	FUNCTION_BLOCK FB 357
	TITLE =G257M COOLING / HEATING GERM 8
	//COPYRIGHT:    (C) 2009  BUHLER AG, CH-9240 UZWIL, SWITZERLAND
	//
	//PRODUCT:      WinCoS_BIW01_09
	//
	//TITLE:        COOLING / HEATING GERM 8
	//                Machine group control
	//                Maschinengruppensteuerung
	//
	//--------------------------------------------------------------------------------
	//
	//IDENT:        AUTHOR:             DEPT:                              DATE:
	//
	//P01_FB357.1.0 K.Renz              CSB41                              13.Jan.2010
	//             1st Release
	//
	//--------------------------------------------------------------------------------
	//
	//PURPOSE:
	//
	//MANUAL :
	//
	//RESTRICTIONS:
	//
	//--------------------------------------------------------------------------------
	AUTHOR  : KR
	FAMILY  : USW
	VERSION : 9.9


	VAR
	  Gr       : FB10;	//Standard interface to group
	  InOutValue1    : DINT; //Data for user
	  InOutValue2    : DINT; //Data for user
	  OutWayConflict : BOOL;	//Data for user
	  OutSelectionOk : BOOL;	//Data for user
	  CmdNewValue : BOOL;	//Data for user
	  CmdNewJob   : BOOL;	//Data for user
	  OutCodeOK   : BOOL;	//Data for user
	  InEndOfJob  : BOOL ;	//Data for user
	  staWayOk      : BOOL ;	//Data for user
	  EdgeStartRelease : BOOL ;	//Data for user
	  USW8  : BOOL;	//Data for user
	  USW9 : BOOL;	//Data for user
	  USW10: BOOL;	//Data for user
	  USW11: BOOL;	//Data for user
	  USW12: BOOL;	//Data for user
	  USW13: BOOL;	//Data for user
	  USW14: BOOL;	//Data for user
	  USW15: BOOL;	//Data for user
	     #A_2845_QXV21 : FB12;   // Motor
	     #A_2845_QXV21AI : FB19;   // AnaInp
	     #A_2845_QXV21AO : FB17;   // AnaOutp
	     #A_2845_QXV21I1 : FB14;   // DigInpCont
	     #A_2845_QXV21I2 : FB14;   // DigInpCont
	     #A_2845_QXV31 : FB12;   // Motor
	     #A_2845_QXV31AI : FB19;   // AnaInp
	     #A_2845_QXV31AO : FB17;   // AnaOutp
	     #A_2845_QXV31I1 : FB14;   // DigInpCont
	     #A_2845_QXV31I2 : FB14;   // DigInpCont
	     #A_2854_MXZ01 : FB12;   // Motor
	     #A_2855_MXZ01 : FB12;   // Motor
	END_VAR
	VAR_TEMP
	   tmpEnable		: BOOL;
	   tmpFlag  		: BOOL;
	   tmpCmdNext		: BOOL;
	   tmpLocal  		: BOOL;
	   tmpAspOk  		: BOOL;
	   tmpHWStop 		: BOOL;
	   tmpInstanzDBNo       : INT ;
	END_VAR
	BEGIN
	NETWORK
	TITLE =
	NETWORK
	TITLE =Read command from group control
	//Parameter
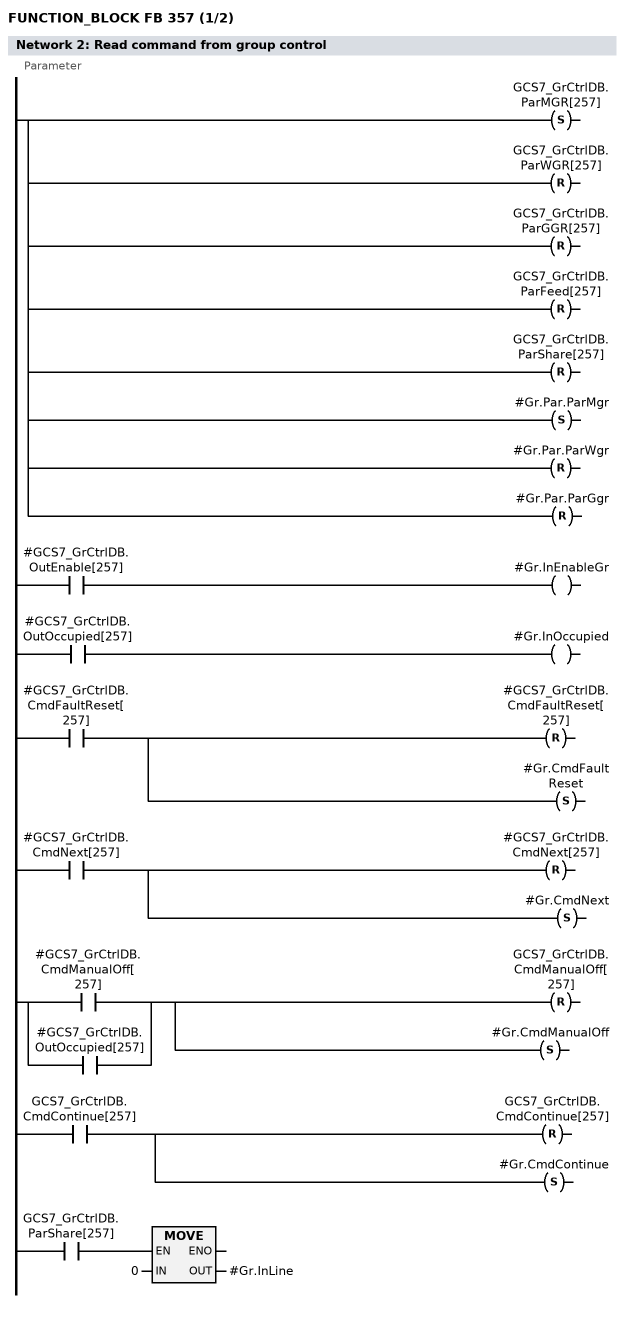
	      SET;
	      S   GCS7_GrCtrlDB.ParMGR[257];
	      R   GCS7_GrCtrlDB.ParWGR[257];
	      R   GCS7_GrCtrlDB.ParGGR[257];
	      R   GCS7_GrCtrlDB.ParFeed[257];
	      R   GCS7_GrCtrlDB.ParShare[257];
	      S   #Gr.Par.ParMgr;
	      R   #Gr.Par.ParWgr;
	      R   #Gr.Par.ParGgr;
	//Command
	      U   #GCS7_GrCtrlDB.OutEnable[257];
	      =   #Gr.InEnableGr;
	      U   #GCS7_GrCtrlDB.OutOccupied[257];
	      =   #Gr.InOccupied;
	      U   #GCS7_GrCtrlDB.CmdFaultReset[257];
	      R   #GCS7_GrCtrlDB.CmdFaultReset[257];
	      S   #Gr.CmdFaultReset;
	      U  #GCS7_GrCtrlDB.CmdNext[257];
	      R   #GCS7_GrCtrlDB.CmdNext[257];
	      S   #Gr.CmdNext;
	      U   #GCS7_GrCtrlDB.CmdManualOff[257];
	      O   #GCS7_GrCtrlDB.OutOccupied[257];
	      R   GCS7_GrCtrlDB.CmdManualOff[257];
	      S   #Gr.CmdManualOff;
	      U  GCS7_GrCtrlDB.CmdContinue[257];
	      R   GCS7_GrCtrlDB.CmdContinue[257];
	      S   #Gr.CmdContinue;
	//Init Line Number
	      U   GCS7_GrCtrlDB.ParShare[257];
	      SPBN WE00;
	      L     0;
	      T     #Gr.InLine;
	WE00: NOP   0;
	NETWORK
	TITLE =Call Methode Control
	// 1. Handle Interface PCControl
	// 2. Prepare mode --> ModePassive,ModeActive,ModeIdling
	// 3. Reset global flags of the group
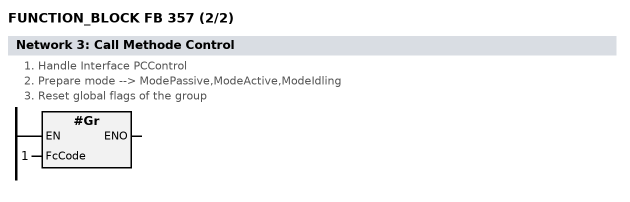
	      CALL #Gr (
	           FcCode                   := 1);
	NETWORK
	TITLE =Restart Idling Time
		L  #Gr.Par.ParIdling;
		L  2;
		>=I;
		SPB IdTm;
		T  #Gr.Par.ParIdling;
	IdTm:   NOP 0;
	      CLR;
	      S    #Gr.CmdRestartIdling;
	NETWORK
	TITLE =Prepare global flags
	NETWORK
	TITLE =Set Pattern (Target position)
	NETWORK
	TITLE =Interlocking WayOk
	//
	NETWORK
	TITLE =Interlocking Autostart
		CLR;
		R   #Gr.OutAutostart;
	NETWORK
	TITLE =Interlocking Enable
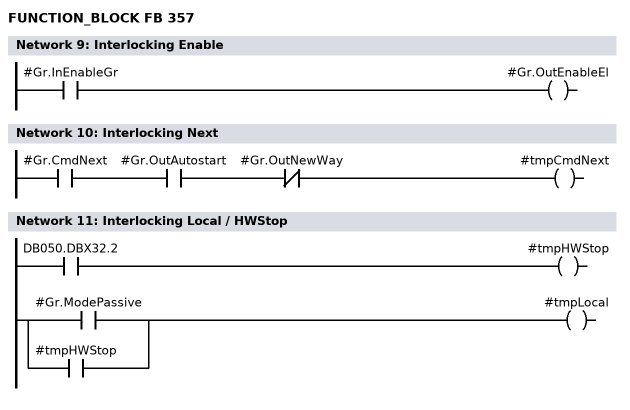
	      U     #Gr.InEnableGr;
	      =     #Gr.OutEnableEl;

	NETWORK
	TITLE =Interlocking Next
	      U     #Gr.CmdNext;
	      U     #Gr.OutAutostart;
	      UN    #Gr.OutNewWay;
	      =    #tmpCmdNext;

	NETWORK
	TITLE =Interlocking Local / HWStop
	      U    DB050.DBX32.2;
	      =    #tmpHWStop;

	      U    #Gr.ModePassive;
	      O    #tmpHWStop;
	      =    #tmpLocal;

	NETWORK
	TITLE =Interlocking Start Warning
	      NOP 0;
	//- Restart after fault --
	      U     #Gr.CmdFaultReset;
	      U     #Gr.VarFault;
	      S       "SYS_StartWarningDB".Area[9].CmdResetStartWarning;
	//- Run Timer --
	      AUF "G257M";
	      CALL  FB100 , DB100(
	       InModeHigher :=FALSE,
	       InArea     :=9,
	       InEnable   :=#Gr.OutEnableEl,
	       InLocal    :=#tmpLocal,
	       InStarted  :=#Gr.VarStarted,
	       InCmdNext  :=#tmpCmdNext,
	       OutCmdNext :=#tmpCmdNext,
	       OutStartwarning:=#Gr.VarStartWarning);
	//- Store Startwarning done  --
	//- Reset Autostart --
	      U     "SYS_StartWarningDB".TmpArea.OutStartReleaseRunningL;
	      FN    #EdgeStartRelease;
	      U     #Gr.VarFault;
	      R     #Gr.OutAutostart;
	NETWORK
	TITLE ==A-2845-QXV21 : RUNNING COOLING UNIT 1 GERMINATING
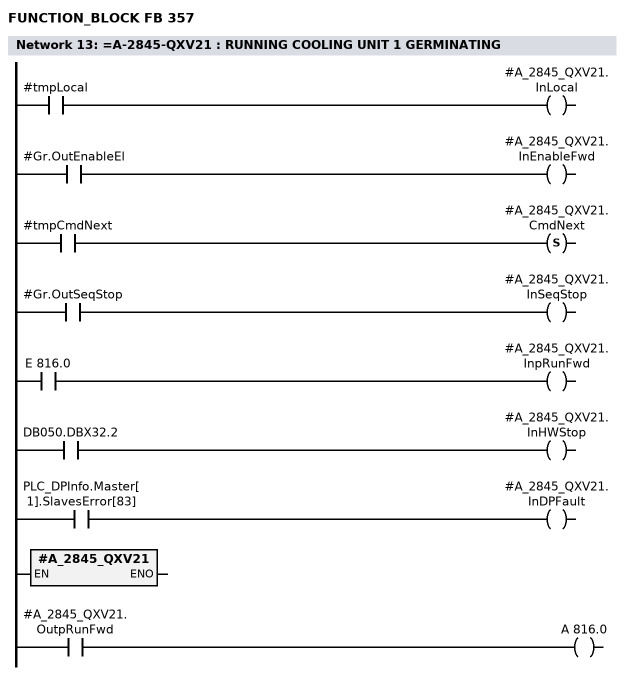
	NOP 0;
	//-InLocal---
	      U     #tmpLocal;
	      =     #A_2845_QXV21.InLocal;
	//
	//-Interlocking---
	      U     #Gr.OutEnableEl;
	      =     #A_2845_QXV21.InEnableFwd;
	//
	      U    #tmpCmdNext;
	      S     #A_2845_QXV21.CmdNext;
	//
	      U     #Gr.OutSeqStop;
	      =     #A_2845_QXV21.InSeqStop;
	//
	//-Read inputs---
	      U     E 816.0;
	      =     #A_2845_QXV21.InpRunFwd;
	      U   DB050.DBX32.2;
	      =     #A_2845_QXV21.InHWStop;
	       U     PLC_DPInfo.Master[1].SlavesError[83];
	       =       #A_2845_QXV21.InDPFault;
	//
	//-Set Parameters---
	//
	//-Call object control---
	      CALL  #A_2845_QXV21;
	//
	//-Write outputs---
	      U     #A_2845_QXV21.OutpRunFwd;
	      =     A 816.0;
	NETWORK
	TITLE ==A-2845-QXV21AI : REGULATING VALVE 1 ACTUAL VALUE
	NOP 0;
	//-InLocal---
	      U     #tmpLocal;
	      =     #A_2845_QXV21AI.InLocal;
	//
	//-Monitoring---
	      CLR;
	      =     #A_2845_QXV21AI.InMonLL;
	      CLR;
	      =     #A_2845_QXV21AI.InMonL;
	      CLR;
	      =     #A_2845_QXV21AI.InMonMid;
	      CLR;
	      =     #A_2845_QXV21AI.InMonH;
	      CLR;
	      =     #A_2845_QXV21AI.InMonHH;
	//
	//-Read inputs---
	      L     PEW872;
	      T     #A_2845_QXV21AI.InpValue;
	      U   DB050.DBX32.2;
	      =     #A_2845_QXV21AI.InHWStop;
	       U     PLC_DPInfo.Master[1].SlavesError[83];
	       =       #A_2845_QXV21AI.InDPFault;
	//
	//-Set Parameters---
	//
	//-Call object control---
	      CALL  #A_2845_QXV21AI;
	//
	//-Write outputs---
	NETWORK
	TITLE ==A-2845-QXV21AO : REGULATING VALVE 1 SET POINT
	NOP 0;
	//-InLocal---
	      U     #tmpLocal;
	      =     #A_2845_QXV21AO.InLocal;
	//
	//-Interlocking---
	      CLR;
	      =     #A_2845_QXV21AO.InDisable;
	//
	//-Values and parameters---
	      L     0;
	      T     #A_2845_QXV21AO.InOutValuePc;
	//
	//-Read inputs---
	      U   DB050.DBX32.2;
	      =     #A_2845_QXV21AO.InHWStop;
	       U     PLC_DPInfo.Master[1].SlavesError[83];
	       =       #A_2845_QXV21AO.InDPFault;
	//
	//-Set Parameters---
	//
	//-Call object control---
	      CALL  #A_2845_QXV21AO;
	//
	//-Write outputs---
	      L     #A_2845_QXV21AO.OutpValue;
	      T     PAW868;
	     UN   "PLC_SystemDB".TestFunctions.StaIOSimuli;
	     SPB PA0;
	      T     AW868;
	      PA0: NOP 0;
	NETWORK
	TITLE ==A-2845-QXV21I1 : REGULATING VALVE 1 CLOSED
	NOP 0;
	//-InLocal---
	      U     #tmpLocal;
	      =     #A_2845_QXV21I1.InLocal;
	//
	//-Monitoring---
	      CLR;
	      =      #A_2845_QXV21I1.InMonTrue;
	      CLR;
	      =      #A_2845_QXV21I1.InMonFalse;
	//
	//-PreAlarm---
	      CLR;
	      =      #A_2845_QXV21I1.InPreAlarmTrue;
	      CLR;
	      =      #A_2845_QXV21I1.InPreAlarmFalse;
	//
	//-Additional commands---
	//      CLR
	//      S     #A_2845_QXV21I1.CmdRunTimeOutTime
	//
	//-Read inputs---
	      U   DB050.DBX32.2;
	      =     #A_2845_QXV21I1.InHWStop;
	//
	//-Set Parameters---
	//
	//-Call object control---
	      CALL  #A_2845_QXV21I1;
	//
	//-Write outputs---
	NETWORK
	TITLE ==A-2845-QXV21I2 : REGULATING VALVE 1 OPENED
	NOP 0;
	//-InLocal---
	      U     #tmpLocal;
	      =     #A_2845_QXV21I2.InLocal;
	//
	//-Monitoring---
	      CLR;
	      =      #A_2845_QXV21I2.InMonTrue;
	      CLR;
	      =      #A_2845_QXV21I2.InMonFalse;
	//
	//-PreAlarm---
	      CLR;
	      =      #A_2845_QXV21I2.InPreAlarmTrue;
	      CLR;
	      =      #A_2845_QXV21I2.InPreAlarmFalse;
	//
	//-Additional commands---
	//      CLR
	//      S     #A_2845_QXV21I2.CmdRunTimeOutTime
	//
	//-Read inputs---
	      U   DB050.DBX32.2;
	      =     #A_2845_QXV21I2.InHWStop;
	//
	//-Set Parameters---
	//
	//-Call object control---
	      CALL  #A_2845_QXV21I2;
	//
	//-Write outputs---
	NETWORK
	TITLE ==A-2845-QXV31 : RUNNING COOLING UNIT 2 GERMINATING
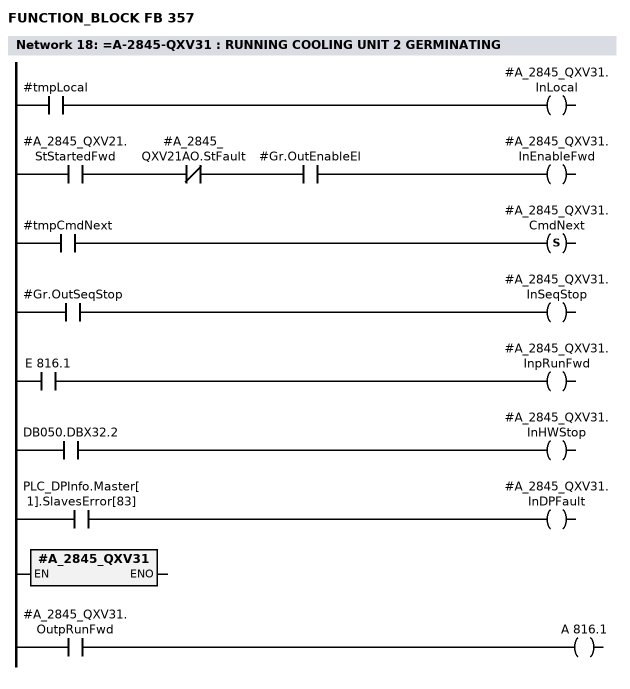
	NOP 0;
	//-InLocal---
	      U     #tmpLocal;
	      =     #A_2845_QXV31.InLocal;
	//
	//-Interlocking---
	      U     #A_2845_QXV21.StStartedFwd;
	      UN    #A_2845_QXV21AO.StFault;
	      U     #Gr.OutEnableEl;
	      =     #A_2845_QXV31.InEnableFwd;
	//
	      U    #tmpCmdNext;
	      S     #A_2845_QXV31.CmdNext;
	//
	      U     #Gr.OutSeqStop;
	      =     #A_2845_QXV31.InSeqStop;
	//
	//-Read inputs---
	      U     E 816.1;
	      =     #A_2845_QXV31.InpRunFwd;
	      U   DB050.DBX32.2;
	      =     #A_2845_QXV31.InHWStop;
	       U     PLC_DPInfo.Master[1].SlavesError[83];
	       =       #A_2845_QXV31.InDPFault;
	//
	//-Set Parameters---
	//
	//-Call object control---
	      CALL  #A_2845_QXV31;
	//
	//-Write outputs---
	      U     #A_2845_QXV31.OutpRunFwd;
	      =     A 816.1;
	NETWORK
	TITLE ==A-2845-QXV31AI : REGULATING VALVE 2 ACTUAL VALUE
	NOP 0;
	//-InLocal---
	      U     #tmpLocal;
	      =     #A_2845_QXV31AI.InLocal;
	//
	//-Monitoring---
	      CLR;
	      =     #A_2845_QXV31AI.InMonLL;
	      CLR;
	      =     #A_2845_QXV31AI.InMonL;
	      CLR;
	      =     #A_2845_QXV31AI.InMonMid;
	      CLR;
	      =     #A_2845_QXV31AI.InMonH;
	      CLR;
	      =     #A_2845_QXV31AI.InMonHH;
	//
	//-Read inputs---
	      L     PEW874;
	      T     #A_2845_QXV31AI.InpValue;
	      U   DB050.DBX32.2;
	      =     #A_2845_QXV31AI.InHWStop;
	       U     PLC_DPInfo.Master[1].SlavesError[83];
	       =       #A_2845_QXV31AI.InDPFault;
	//
	//-Set Parameters---
	//
	//-Call object control---
	      CALL  #A_2845_QXV31AI;
	//
	//-Write outputs---
	NETWORK
	TITLE ==A-2845-QXV31AO : REGULATING VALVE 2 SET POINT
	NOP 0;
	//-InLocal---
	      U     #tmpLocal;
	      =     #A_2845_QXV31AO.InLocal;
	//
	//-Interlocking---
	      CLR;
	      =     #A_2845_QXV31AO.InDisable;
	//
	//-Values and parameters---
	      L     0;
	      T     #A_2845_QXV31AO.InOutValuePc;
	//
	//-Read inputs---
	      U   DB050.DBX32.2;
	      =     #A_2845_QXV31AO.InHWStop;
	       U     PLC_DPInfo.Master[1].SlavesError[83];
	       =       #A_2845_QXV31AO.InDPFault;
	//
	//-Set Parameters---
	//
	//-Call object control---
	      CALL  #A_2845_QXV31AO;
	//
	//-Write outputs---
	      L     #A_2845_QXV31AO.OutpValue;
	      T     PAW870;
	     UN   "PLC_SystemDB".TestFunctions.StaIOSimuli;
	     SPB PA1;
	      T     AW870;
	      PA1: NOP 0;
	NETWORK
	TITLE ==A-2845-QXV31I1 : REGULATING VALVE 2 CLOSED
	NOP 0;
	//-InLocal---
	      U     #tmpLocal;
	      =     #A_2845_QXV31I1.InLocal;
	//
	//-Monitoring---
	      CLR;
	      =      #A_2845_QXV31I1.InMonTrue;
	      CLR;
	      =      #A_2845_QXV31I1.InMonFalse;
	//
	//-PreAlarm---
	      CLR;
	      =      #A_2845_QXV31I1.InPreAlarmTrue;
	      CLR;
	      =      #A_2845_QXV31I1.InPreAlarmFalse;
	//
	//-Additional commands---
	//      CLR
	//      S     #A_2845_QXV31I1.CmdRunTimeOutTime
	//
	//-Read inputs---
	      U   DB050.DBX32.2;
	      =     #A_2845_QXV31I1.InHWStop;
	//
	//-Set Parameters---
	//
	//-Call object control---
	      CALL  #A_2845_QXV31I1;
	//
	//-Write outputs---
	NETWORK
	TITLE ==A-2845-QXV31I2 : REGULATING VALVE 2 OPENED
	NOP 0;
	//-InLocal---
	      U     #tmpLocal;
	      =     #A_2845_QXV31I2.InLocal;
	//
	//-Monitoring---
	      CLR;
	      =      #A_2845_QXV31I2.InMonTrue;
	      CLR;
	      =      #A_2845_QXV31I2.InMonFalse;
	//
	//-PreAlarm---
	      CLR;
	      =      #A_2845_QXV31I2.InPreAlarmTrue;
	      CLR;
	      =      #A_2845_QXV31I2.InPreAlarmFalse;
	//
	//-Additional commands---
	//      CLR
	//      S     #A_2845_QXV31I2.CmdRunTimeOutTime
	//
	//-Read inputs---
	      U   DB050.DBX32.2;
	      =     #A_2845_QXV31I2.InHWStop;
	//
	//-Set Parameters---
	//
	//-Call object control---
	      CALL  #A_2845_QXV31I2;
	//
	//-Write outputs---
	NETWORK
	TITLE ==A-2854-MXZ01 : WATER PUMP 1
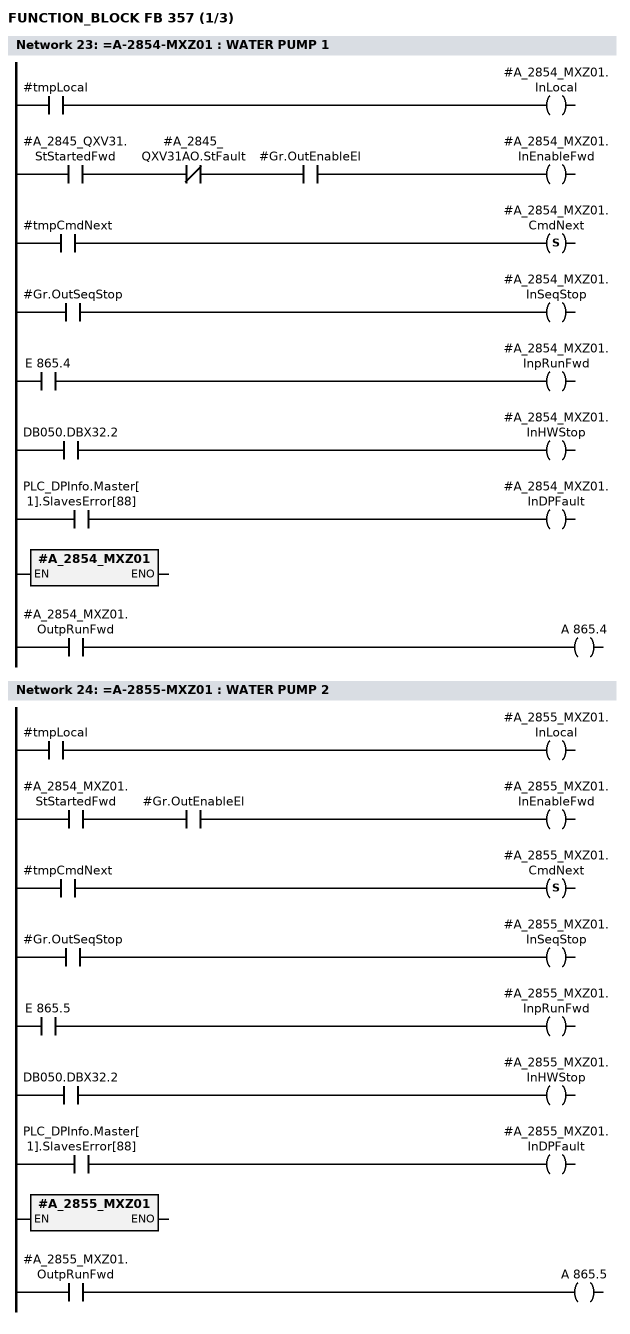
	NOP 0;
	//-InLocal---
	      U     #tmpLocal;
	      =     #A_2854_MXZ01.InLocal;
	//
	//-Interlocking---
	      U     #A_2845_QXV31.StStartedFwd;
	      UN    #A_2845_QXV31AO.StFault;
	      U     #Gr.OutEnableEl;
	      =     #A_2854_MXZ01.InEnableFwd;
	//
	      U    #tmpCmdNext;
	      S     #A_2854_MXZ01.CmdNext;
	//
	      U     #Gr.OutSeqStop;
	      =     #A_2854_MXZ01.InSeqStop;
	//
	//-Read inputs---
	      U     E 865.4;
	      =     #A_2854_MXZ01.InpRunFwd;
	      U   DB050.DBX32.2;
	      =     #A_2854_MXZ01.InHWStop;
	       U     PLC_DPInfo.Master[1].SlavesError[88];
	       =       #A_2854_MXZ01.InDPFault;
	//
	//-Set Parameters---
	//
	//-Call object control---
	      CALL  #A_2854_MXZ01;
	//
	//-Write outputs---
	      U     #A_2854_MXZ01.OutpRunFwd;
	      =     A 865.4;
	NETWORK
	TITLE ==A-2855-MXZ01 : WATER PUMP 2
	NOP 0;
	//-InLocal---
	      U     #tmpLocal;
	      =     #A_2855_MXZ01.InLocal;
	//
	//-Interlocking---
	      U     #A_2854_MXZ01.StStartedFwd;
	      U     #Gr.OutEnableEl;
	      =     #A_2855_MXZ01.InEnableFwd;
	//
	      U    #tmpCmdNext;
	      S     #A_2855_MXZ01.CmdNext;
	//
	      U     #Gr.OutSeqStop;
	      =     #A_2855_MXZ01.InSeqStop;
	//
	//-Read inputs---
	      U     E 865.5;
	      =     #A_2855_MXZ01.InpRunFwd;
	      U   DB050.DBX32.2;
	      =     #A_2855_MXZ01.InHWStop;
	       U     PLC_DPInfo.Master[1].SlavesError[88];
	       =       #A_2855_MXZ01.InDPFault;
	//
	//-Set Parameters---
	//
	//-Call object control---
	      CALL  #A_2855_MXZ01;
	//
	//-Write outputs---
	      U     #A_2855_MXZ01.OutpRunFwd;
	      =     A 865.5;
	NETWORK
	TITLE =Test Fault
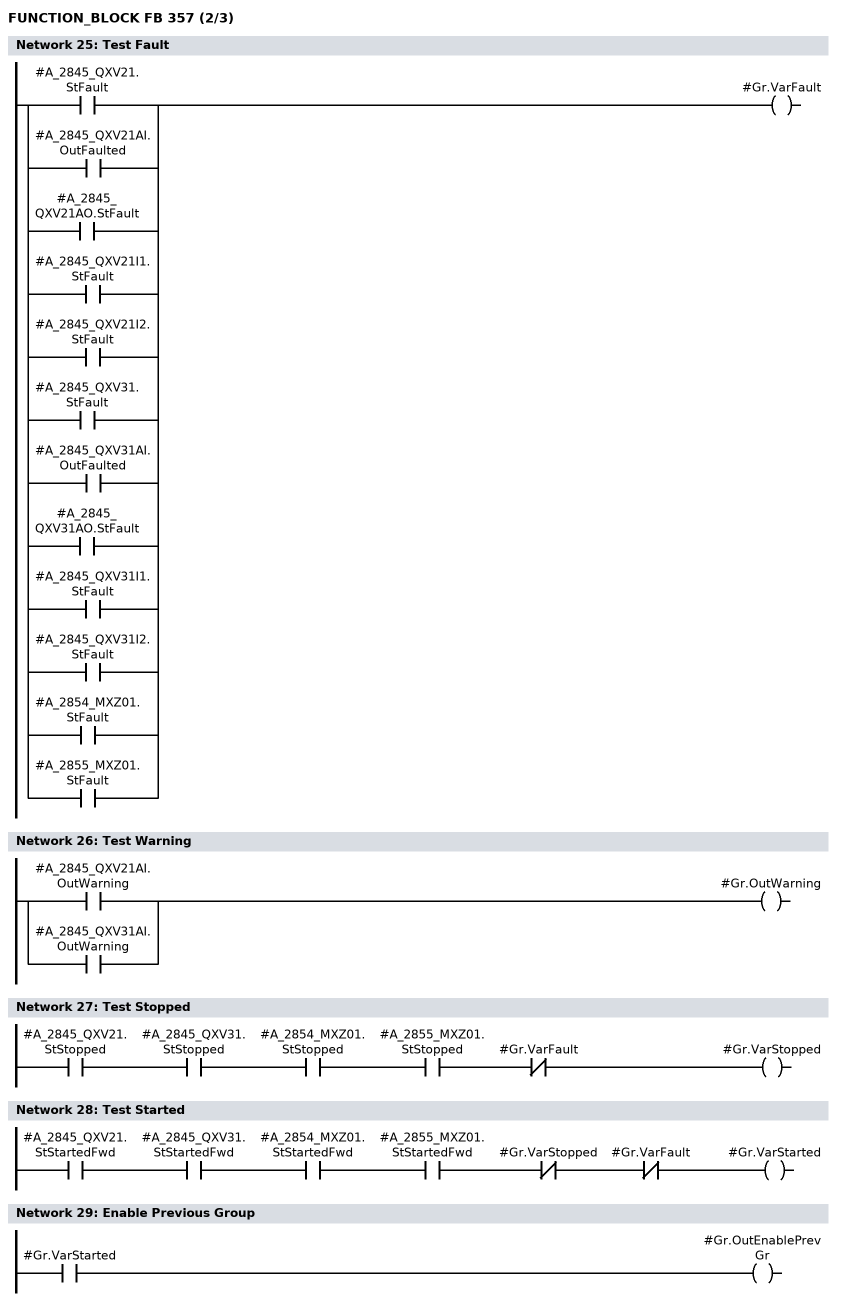
	      U     #A_2845_QXV21.StFault;
	      O     #A_2845_QXV21AI.OutFaulted;
	      O     #A_2845_QXV21AO.StFault;
	      O     #A_2845_QXV21I1.StFault;
	      O     #A_2845_QXV21I2.StFault;
	      O     #A_2845_QXV31.StFault;
	      O     #A_2845_QXV31AI.OutFaulted;
	      O     #A_2845_QXV31AO.StFault;
	      O     #A_2845_QXV31I1.StFault;
	      O     #A_2845_QXV31I2.StFault;
	      O     #A_2854_MXZ01.StFault;
	      O     #A_2855_MXZ01.StFault;
	      =     #Gr.VarFault;
	NETWORK
	TITLE =Test Warning
	      U     #A_2845_QXV21AI.OutWarning;
	      O     #A_2845_QXV31AI.OutWarning;
	      =     #Gr.OutWarning;
	NETWORK
	TITLE =Test Stopped
	      U     #A_2845_QXV21.StStopped;
	      U     #A_2845_QXV31.StStopped;
	      U     #A_2854_MXZ01.StStopped;
	      U     #A_2855_MXZ01.StStopped;
	      UN   #Gr.VarFault;
	      =     #Gr.VarStopped;
	NETWORK
	TITLE =Test Started
	      U     #A_2845_QXV21.StStartedFwd;
	      U     #A_2845_QXV31.StStartedFwd;
	      U     #A_2854_MXZ01.StStartedFwd;
	      U     #A_2855_MXZ01.StStartedFwd;
	      UN  #Gr.VarStopped;
	      UN  #Gr.VarFault;
	      =     #Gr.VarStarted;
	NETWORK
	TITLE =Enable Previous Group
	      U    #Gr.VarStarted;
	      =     #Gr.OutEnablePrevGr;
	NETWORK
	TITLE =Call Methode State
	//1. Make State of the group: This function use the signals:
	//        Gr.VarStopped, Gr.VarStarted, Gr.VarFault
	//2.Reset Commands to group: e.g.CmdFaultReset
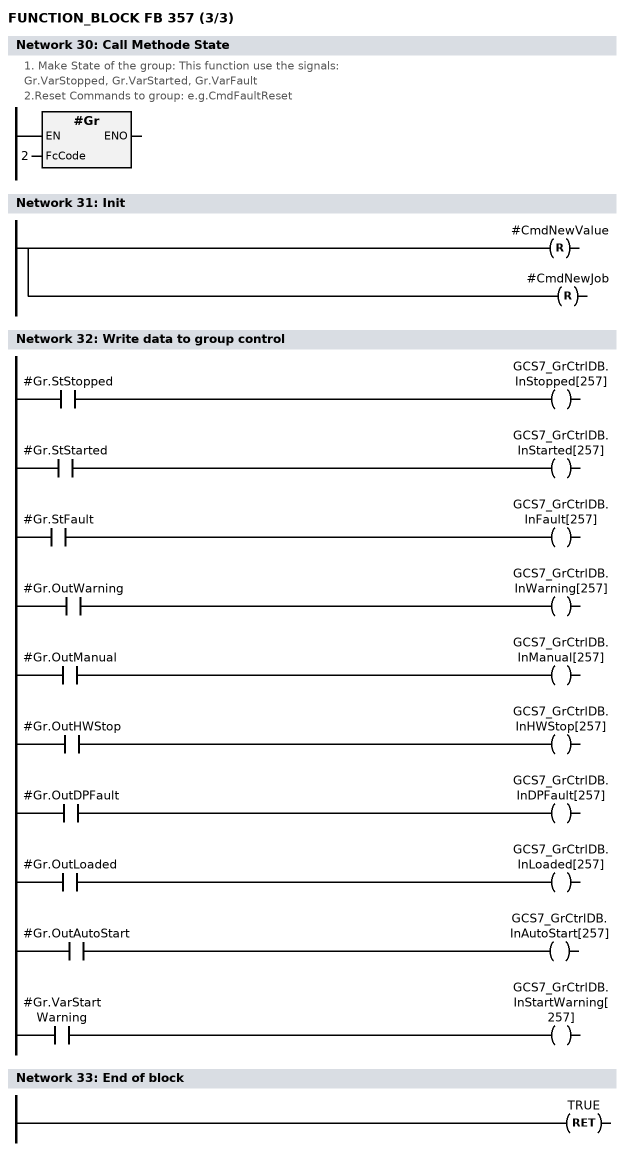
	      CALL #Gr (
	           FcCode                   := 2);
	NETWORK
	TITLE =Init
	      SET;
	      R    #CmdNewValue;
	      R    #CmdNewJob;
	NETWORK
	TITLE =Write data to group control
	      U   #Gr.StStopped;
	      =   GCS7_GrCtrlDB.InStopped[257];
	      U   #Gr.StStarted;
	      =   GCS7_GrCtrlDB.InStarted[257];
	      U   #Gr.StFault;
	      =   GCS7_GrCtrlDB.InFault[257];
	      U   #Gr.OutWarning;
	      =   GCS7_GrCtrlDB.InWarning[257];
	      U   #Gr.OutManual;
	      =   GCS7_GrCtrlDB.InManual[257];
	      U   #Gr.OutHWStop;
	      =   GCS7_GrCtrlDB.InHWStop[257];
	      U   #Gr.OutDPFault;
	      =   GCS7_GrCtrlDB.InDPFault[257];
	      U   #Gr.OutLoaded;
	      =   GCS7_GrCtrlDB.InLoaded[257];
	      U   #Gr.OutAutoStart;
	      =   GCS7_GrCtrlDB.InAutoStart[257];
	      U   #Gr.VarStartWarning;
	      =   GCS7_GrCtrlDB.InStartWarning[257];
	NETWORK
	TITLE =End of block

	BE

	END_FUNCTION_BLOCK
